FUNCTION_BLOCK Test_TStreamAddReadArgType EXTENDS T_UnitTestBase
VAR
    Stream : T_Stream(StreamLength := 2);
END_VAR

{attribute 'analysis' := '-33'} // inhibit unused variable warning
METHOD RunTest
IF Retest THEN
    SUPER^.Init();
END_IF

IF TestCompleted THEN
    RETURN;
END_IF

F_Inc(CycleCount);
IF CycleCount > 1000 THEN
    Fail(Message := 'Timeout');
END_IF

Stream.Init(2);

Stream.SetNextArgTypeId(E_ArgTypeId.Type_LINT);

AssertEquals_UDINT(Expected     := 2,
                             Actual       := Stream.WritePosition,
                             Message := 'Stream.WritePosition');

Stream.SetReadPosition(0);

AssertEquals_INT(Expected     := E_ArgTypeId.Type_LINT,
                           Actual       := Stream.GetNextArgTypeId(),
                           Message := 'Stream.GetNextArgTypeId()');

AssertEquals_UDINT(Expected     := 2,
                             Actual       := Stream.ReadPosition,
                             Message := 'Stream.ReadPosition');

TestCompleted := TRUE;
END_METHOD

END_FUNCTION_BLOCK

(* stored: Version 1.1.0.1, ProductVersion 3.1.4024.15
   POU Test_TStreamAddReadArgType: Id {3f884bce-15bd-4284-8d11-76cd93e31e35}, SpecialFunc None
   Method RunTest: Id {f22959de-fa1e-47c4-89cc-d8ee70c8e77d} *)
